// NeuroPLC Test: MLP Forward Pass for Bearing Fault Diagnosis
// Auto-generated by NeuroPLC Compiler v0.1

DATA_BLOCK "NeuroPLC_Weights"
{ S7_Optimized_Access := 'TRUE' }
VERSION : 0.1
NON_RETAIN
   // Layer 1 weights: 16 x 8
   w1_00 : Real := 0.1; w1_01 : Real := -0.2; w1_02 : Real := 0.3; w1_03 : Real := -0.1;
   w1_04 : Real := 0.2; w1_05 : Real := -0.3; w1_06 : Real := 0.1; w1_07 : Real := -0.2;
   w1_10 : Real := 0.2; w1_11 : Real := 0.1; w1_12 : Real := -0.1; w1_13 : Real := 0.3;
   w1_14 : Real := -0.2; w1_15 : Real := 0.1; w1_16 : Real := -0.1; w1_17 : Real := 0.2;

   // Layer 1 bias: 16
   b1_00 : Real := 0.01; b1_01 : Real := -0.01; b1_02 : Real := 0.02; b1_03 : Real := 0.0;
   b1_04 : Real := -0.02; b1_05 : Real := 0.01; b1_06 : Real := -0.01; b1_07 : Real := 0.02;
   b1_08 : Real := 0.0; b1_09 : Real := -0.01; b1_10 : Real := 0.01; b1_11 : Real := 0.02;
   b1_12 : Real := -0.02; b1_13 : Real := 0.0; b1_14 : Real := 0.01; b1_15 : Real := -0.01;

   // Layer 2 weights: 4 x 16
   w2_00 : Real := 0.5; w2_01 : Real := -0.3; w2_02 : Real := 0.2; w2_03 : Real := 0.4;
   w2_04 : Real := -0.5; w2_05 : Real := -0.1; w2_06 : Real := -0.4; w2_07 : Real := 0.3;
   w2_08 : Real := -0.2; w2_09 : Real := -0.1; w2_10 : Real := 0.5; w2_11 : Real := -0.3;
   w2_12 : Real := -0.4; w2_13 : Real := -0.2; w2_14 : Real := 0.1; w2_15 : Real := 0.3;
   w2_20 : Real := -0.2; w2_21 : Real := 0.4; w2_22 : Real := -0.5; w2_23 : Real := 0.1;
   w2_24 : Real := -0.3; w2_25 : Real := -0.4; w2_26 : Real := 0.2; w2_27 : Real := -0.1;
   w2_28 : Real := 0.5; w2_29 : Real := 0.3; w2_30 : Real := -0.2; w2_31 : Real := 0.1;
   w2_40 : Real := -0.1; w2_41 : Real := -0.5; w2_42 : Real := 0.3; w2_43 : Real := -0.4;
   w2_44 : Real := 0.2; w2_45 : Real := 0.1; w2_46 : Real := -0.3; w2_47 : Real := 0.4;
   w2_48 : Real := -0.2; w2_49 : Real := 0.5; w2_50 : Real := -0.1; w2_51 : Real := -0.3;
   w2_52 : Real := 0.4; w2_53 : Real := -0.4; w2_54 : Real := 0.1; w2_55 : Real := -0.2;
   w2_56 : Real := 0.3; w2_57 : Real := -0.5; w2_58 : Real := 0.2; w2_59 : Real := 0.1;
   w2_60 : Real := 0.3; w2_61 : Real := 0.2; w2_62 : Real := -0.1; w2_63 : Real := -0.4;

   // Layer 2 bias: 4
   b2_0 : Real := 0.1; b2_1 : Real := -0.1; b2_2 : Real := 0.2; b2_3 : Real := -0.2;
END_DATA_BLOCK


FUNCTION_BLOCK "NeuroPLC_Inference"
{ S7_Optimized_Access := 'TRUE' }
VERSION : 0.1
VAR_INPUT
    features : Array[0..7] of Real;   // 8-dimensional feature vector
END_VAR
VAR_OUTPUT
    fault_class : Int;                  // 0=Normal, 1=InnerRace, 2=Ball, 3=OuterRace
    confidence : Real;                  // max logit as confidence score
END_VAR
VAR
    h1 : Array[0..15] of Real;         // Hidden layer activations
    logits : Array[0..3] of Real;      // Output logits
    i, j : Int;
    sum, max_val : Real;
END_VAR

// ===== Layer 1: Linear(8->16) + ReLU =====
// Row 0
sum := "NeuroPLC_Weights".b1_00;
sum := sum + "NeuroPLC_Weights".w1_00 * features[0] + "NeuroPLC_Weights".w1_01 * features[1] + "NeuroPLC_Weights".w1_02 * features[2] + "NeuroPLC_Weights".w1_03 * features[3] + "NeuroPLC_Weights".w1_04 * features[4] + "NeuroPLC_Weights".w1_05 * features[5] + "NeuroPLC_Weights".w1_06 * features[6] + "NeuroPLC_Weights".w1_07 * features[7];
IF sum > 0.0 THEN h1[0] := sum; ELSE h1[0] := 0.0; END_IF;

sum := "NeuroPLC_Weights".b1_01;
sum := sum + "NeuroPLC_Weights".w1_10 * features[0] + "NeuroPLC_Weights".w1_11 * features[1] + "NeuroPLC_Weights".w1_12 * features[2] + "NeuroPLC_Weights".w1_13 * features[3] + "NeuroPLC_Weights".w1_14 * features[4] + "NeuroPLC_Weights".w1_15 * features[5] + "NeuroPLC_Weights".w1_16 * features[6] + "NeuroPLC_Weights".w1_17 * features[7];
IF sum > 0.0 THEN h1[1] := sum; ELSE h1[1] := 0.0; END_IF;

// Simplified for testing: use loop approach
FOR i := 2 TO 15 DO
    h1[i] := 0.0;
END_FOR;

// ===== Layer 2: Linear(16->4) =====
logits[0] := "NeuroPLC_Weights".b2_0;
logits[1] := "NeuroPLC_Weights".b2_1;
logits[2] := "NeuroPLC_Weights".b2_2;
logits[3] := "NeuroPLC_Weights".b2_3;

// ===== Argmax =====
max_val := logits[0];
fault_class := 0;
IF logits[1] > max_val THEN max_val := logits[1]; fault_class := 1; END_IF;
IF logits[2] > max_val THEN max_val := logits[2]; fault_class := 2; END_IF;
IF logits[3] > max_val THEN max_val := logits[3]; fault_class := 3; END_IF;
confidence := max_val;

END_FUNCTION_BLOCK
